// TIA Portal V15.1 export
// export: Created 2024-06-21T08:41:05.5283843Z, ExportSetting WithDefaults, DisplayName Totally Integrated Automation Portal, DisplayVersion V15.1 Update 5, DisplayName TIA Portal Openness, DisplayVersion V15.1 Update 5, DisplayName SINAMICS Startdrive Advanced, DisplayVersion V15.1, DisplayName G130, G150, S120, S150, SINAMICS MV, S210, DisplayVersion V15.1, DisplayName G110M, G120, G120C, G120D, G120P, DisplayVersion V15.1, DisplayName STEP 7 Professional, DisplayVersion V15.1 Update 5, DisplayName STEP 7 Safety, DisplayVersion V15.1, DisplayName WinCC Professional, DisplayVersion V15.1 Update 5, DisplayName SIMATIC Visualization Architect, DisplayVersion V15.1
FUNCTION_BLOCK "LGBMotor2W2S-MoviFitFCPN"   // FB6619, FBD
TITLE = LGBMotor2W2S-MoviFitFCPN
{ S7_Optimized_Access := 'TRUE' }
AUTHOR : ENGIE
FAMILY : Actuator
VERSION : 0.1
// ============================================================================
// This module is used in applications when a Motor 2 way - 2 speed equipped with SEW MOVIFIT FC with fieldbus steering is needed.
// ============================================================================
// stored: AutoNumber false, IsIECCheckEnabled false, IsRetainMemResEnabled false, MemoryReserve 100, SetENOAutomatically False, UDAEnableTagReadback false
   VAR_INPUT
      I_MotorProtection { ExternalAccessible := 'False'; ExternalVisible := 'False'; ExternalWritable := 'False'} : Bool;   // Motor protection
      I_AlarmResetPB { ExternalAccessible := 'False'; ExternalVisible := 'False'; ExternalWritable := 'False'} : Bool;   // Alarm Reset Pushbutton is Activated
      I_SafetyStatusWord { ExternalAccessible := 'False'; ExternalVisible := 'False'; ExternalWritable := 'False'} : Word;   // Safety status word
      I_SafetyControlWord { ExternalAccessible := 'False'; ExternalVisible := 'False'; ExternalWritable := 'False'} : Word;   // Safety control word
      I_SafetyOk { ExternalAccessible := 'False'; ExternalVisible := 'False'; ExternalWritable := 'False'} : Bool;   // Safety ok
      I_MotionStopOk { ExternalAccessible := 'False'; ExternalVisible := 'False'; ExternalWritable := 'False'} : Bool;   // Safety Ok / The motion stop is Ok
      I_LSpdSetMotorCmd { ExternalAccessible := 'False'; ExternalVisible := 'False'; ExternalWritable := 'False'} : Bool;   // Low speed Set Command from function after interlock
      I_HSpdSetMotorCmd { ExternalAccessible := 'False'; ExternalVisible := 'False'; ExternalWritable := 'False'} : Bool;   // High Speed Set Command from function after Interlock
      I_LSpdResMotorCmd { ExternalAccessible := 'False'; ExternalVisible := 'False'; ExternalWritable := 'False'} : Bool;   // Low speed Reset Command from function after interlock
      I_HSpdResMotorCmd { ExternalAccessible := 'False'; ExternalVisible := 'False'; ExternalWritable := 'False'} : Bool;   // High speed Reset Command from function after Interlock
      I_LowSpeed { ExternalAccessible := 'False'; ExternalVisible := 'False'; ExternalWritable := 'False'} : Real;   // Low speed value 0-100%
      I_HighSpeed { ExternalAccessible := 'False'; ExternalVisible := 'False'; ExternalWritable := 'False'} : Real;   // High speed value 0-100%
      I_Ramp { ExternalAccessible := 'False'; ExternalVisible := 'False'; ExternalWritable := 'False'} : Time := T#1s;   // Ramp send in miliseconds (range : 100-10000ms, if 0 then default 1s will be used)
      I_BrakeRelease { ExternalAccessible := 'False'; ExternalVisible := 'False'; ExternalWritable := 'False'} : Bool;   // Command brake release
      I_ParameterSet { ExternalAccessible := 'False'; ExternalVisible := 'False'; ExternalWritable := 'False'} : Bool;   // Select parameter set
   END_VAR
   VAR_OUTPUT
      O_MotorProtectionAlarm { ExternalAccessible := 'False'; ExternalVisible := 'False'; ExternalWritable := 'False'} : Bool;   // Motor protection alarm
      O_SafetySwitchAlarm { ExternalAccessible := 'False'; ExternalVisible := 'False'; ExternalWritable := 'False'} : Bool;   // Safety switch alarm
      O_ConfigRampAlarm { ExternalAccessible := 'False'; ExternalVisible := 'False'; ExternalWritable := 'False'} : Bool;   // Config alarm
      O_ConfigRampCalcAlarm { ExternalAccessible := 'False'; ExternalVisible := 'False'; ExternalWritable := 'False'} : Bool;   // Config alarm
      O_STOAlarm { ExternalAccessible := 'False'; ExternalVisible := 'False'; ExternalWritable := 'False'} : Bool;   // Drive fault / STO alarm
      O_MotionStopWarning { ExternalAccessible := 'False'; ExternalVisible := 'False'; ExternalWritable := 'False'} : Bool;   // Drive fault / Motion Stop warning
      O_DriveFaultAlarm { ExternalAccessible := 'False'; ExternalVisible := 'False'; ExternalWritable := 'False'} : Bool;   // Drive fault
      O_DriveWarning { ExternalAccessible := 'False'; ExternalVisible := 'False'; ExternalWritable := 'False'} : Bool;   // Drive warning
      O_DriveReady { ExternalAccessible := 'False'; ExternalVisible := 'False'; ExternalWritable := 'False'} : Bool;   // Drive ready
      O_PODataNotEnabled { ExternalAccessible := 'False'; ExternalVisible := 'False'; ExternalWritable := 'False'} : Bool;   // Process data is enabled (1 = Drive can be controlled via fieldbus)
      O_ParameterSet { ExternalAccessible := 'False'; ExternalVisible := 'False'; ExternalWritable := 'False'} : Bool;   // Active parameter set
      O_OutputStageEnabled { ExternalAccessible := 'False'; ExternalVisible := 'False'; ExternalWritable := 'False'} : Bool;   // Inverter output stage is enabled
      O_Brake { ExternalAccessible := 'False'; ExternalVisible := 'False'; ExternalWritable := 'False'} : Bool;   // Brake status
      O_AlarmABCondition { ExternalAccessible := 'False'; ExternalVisible := 'False'; ExternalWritable := 'False'} : Bool;   // Alarm AB Condition
   END_VAR
   VAR_IN_OUT
      IO_Modes : "Modes";
      IO_Alarm : "Alarm";
      H_HMI : "H_HMI";
      "H_GBMotor2W2S-MoviFitFCPN" : "H_GBMotor2W2S-MoviFitFCPN";   // HMI UDT
      C_EnableAlarm { ExternalAccessible := 'False'; ExternalVisible := 'False'; ExternalWritable := 'False'} : Bool;   // Enable Alarm
      C_MotorProtectionUsed { ExternalAccessible := 'False'; ExternalVisible := 'False'; ExternalWritable := 'False'} : Bool := True;   // Motor Protection used
      C_MotorProtectionNc { ExternalAccessible := 'False'; ExternalVisible := 'False'; ExternalWritable := 'False'} : Bool := True;   // Motor Protection Normally closed
      C_MotionStopUsed { ExternalAccessible := 'False'; ExternalVisible := 'False'; ExternalWritable := 'False'} : Bool;   // Motion Stop used
      C_HWSubInput { ExternalAccessible := 'False'; ExternalVisible := 'False'; ExternalWritable := 'False'} : HW_SUBMODULE;   // Inputs telegram 3 Hardware identifier
      C_HWSubInputStatus { ExternalAccessible := 'False'; ExternalVisible := 'False'; ExternalWritable := 'False'} : HW_SUBMODULE;   // Status telegram MOVIFIT Hardware identifier
      C_HWSubOutput { ExternalAccessible := 'False'; ExternalVisible := 'False'; ExternalWritable := 'False'} : HW_SUBMODULE;   // Outputs telegram 3 Hardware identifier
      C_InitDirection { ExternalAccessible := 'False'; ExternalVisible := 'False'; ExternalWritable := 'False'} : Bool;   // Initialisation of the direction
      C_DriveCurrent { ExternalAccessible := 'False'; ExternalVisible := 'False'; ExternalWritable := 'False'} : Real;   // Reference current of the drive
      C_MotorCurrent { ExternalAccessible := 'False'; ExternalVisible := 'False'; ExternalWritable := 'False'} : Real;   // Reference current of the motor
      C_MotorRPM { ExternalAccessible := 'False'; ExternalVisible := 'False'; ExternalWritable := 'False'} : Real;   // Reference RPM of the motor
      C_RatioGearbox { ExternalAccessible := 'False'; ExternalVisible := 'False'; ExternalWritable := 'False'} : Real;   // Ratio Gearbox <-> Motor
      C_Diameter { ExternalAccessible := 'False'; ExternalVisible := 'False'; ExternalWritable := 'False'} : Real;   // Diameter in mm
      C_Acceleration { ExternalAccessible := 'False'; ExternalVisible := 'False'; ExternalWritable := 'False'} : Real;   // Acceleration in m/s²
   END_VAR
   VAR
      EnableAlarmHWSR { ExternalAccessible := 'False'; ExternalVisible := 'False'; ExternalWritable := 'False'} : Bool;   // Enable Alarms from the hardware
      EnableAlarmHW { ExternalAccessible := 'False'; ExternalVisible := 'False'; ExternalWritable := 'False'} : Bool;   // Enable Alarms from the hardware
      SetFrequency { ExternalAccessible := 'False'; ExternalVisible := 'False'; ExternalWritable := 'False'} : Real;   // Set frequency dependant on config
      ResFrequency { ExternalAccessible := 'False'; ExternalVisible := 'False'; ExternalWritable := 'False'} : Real;   // Reset frequency dependant on config
      MotorProtectionAlarm { ExternalAccessible := 'False'; ExternalVisible := 'False'; ExternalWritable := 'False'} : Bool;   // Motor protection alarm
      MotorProtectionAlarmABCond { ExternalAccessible := 'False'; ExternalVisible := 'False'; ExternalWritable := 'False'} : Bool;   // Motor protection alarm condition
      SafetySwitchAlarm { ExternalAccessible := 'False'; ExternalVisible := 'False'; ExternalWritable := 'False'} : Bool;   // Safety Switch alarm
      SafetySwitchAlarmABCond { ExternalAccessible := 'False'; ExternalVisible := 'False'; ExternalWritable := 'False'} : Bool;   // Safety Switch alarm condition
      DriveFaultAlarm { ExternalAccessible := 'False'; ExternalVisible := 'False'; ExternalWritable := 'False'} : Bool;   // Drive fault alarm
      DriveFaultAlarmABCond { ExternalAccessible := 'False'; ExternalVisible := 'False'; ExternalWritable := 'False'} : Bool;   // Drive fault alarm condition
      STOAlarm { ExternalAccessible := 'False'; ExternalVisible := 'False'; ExternalWritable := 'False'} : Bool;   // Drive fault alarm / STO feedback fault alarm
      STOAlarmABCond { ExternalAccessible := 'False'; ExternalVisible := 'False'; ExternalWritable := 'False'} : Bool;   // Drive fault alarm condition / STO feedback fault alarm condition
      MotionStopWarning { ExternalAccessible := 'False'; ExternalVisible := 'False'; ExternalWritable := 'False'} : Bool;   // Drive fault alarm / Motion Stop warning
      ConfigRampAlarm { ExternalAccessible := 'False'; ExternalVisible := 'False'; ExternalWritable := 'False'} : Bool;   // Config alarm
      ConfigRampCalcAlarm { ExternalAccessible := 'False'; ExternalVisible := 'False'; ExternalWritable := 'False'} : Bool;   // Config alarm
      Start { ExternalAccessible := 'False'; ExternalVisible := 'False'; ExternalWritable := 'False'} : Bool;   // Start command to drive
      SetpointSpeed { ExternalAccessible := 'False'; ExternalVisible := 'False'; ExternalWritable := 'False'} : Real;   // Setpoint speed
      SetpointSpeedCalc { ExternalAccessible := 'False'; ExternalVisible := 'False'; ExternalWritable := 'False'} : Real;   // Setpoint speed
      OutputStageEnabled { ExternalAccessible := 'False'; ExternalVisible := 'False'; ExternalWritable := 'False'} : Bool;   // Inverter output stage is enabled
      MaintenanceSwitch { ExternalAccessible := 'False'; ExternalVisible := 'False'; ExternalWritable := 'False'} : Bool;   // Maintenance switch activated (1=mains OFF)
      PODataEnabled { ExternalAccessible := 'False'; ExternalVisible := 'False'; ExternalWritable := 'False'} : Bool;   // Process data is enabled (1 = Drive can be controlled via fieldbus)
      PODataDisabled { ExternalAccessible := 'False'; ExternalVisible := 'False'; ExternalWritable := 'False'} : Bool;   // Process data is enabled (1 = Drive can be controlled via fieldbus)
      Fault { ExternalAccessible := 'False'; ExternalVisible := 'False'; ExternalWritable := 'False'} : Bool;   // Fault present
      Brake { ExternalAccessible := 'False'; ExternalVisible := 'False'; ExternalWritable := 'False'} : Bool;   // Brake status
      ActorVoltageOverloadDO00 { ExternalAccessible := 'False'; ExternalVisible := 'False'; ExternalWritable := 'False'} : Bool;   // Short circuit / overload of the actuator voltage for digital output DO00
      ActorVoltageOverloadDO01 { ExternalAccessible := 'False'; ExternalVisible := 'False'; ExternalWritable := 'False'} : Bool;   // Short circuit / overload of the actuator voltage for digital output DO01
      ActorVoltageOverloadDO02 { ExternalAccessible := 'False'; ExternalVisible := 'False'; ExternalWritable := 'False'} : Bool;   // Short circuit / overload of the actuator voltage for digital output DO02
      ActorVoltageOverloadDO03 { ExternalAccessible := 'False'; ExternalVisible := 'False'; ExternalWritable := 'False'} : Bool;   // Short circuit / overload of the actuator voltage for digital output DO03
      SensorVoltageOverloadGroup1 { ExternalAccessible := 'False'; ExternalVisible := 'False'; ExternalWritable := 'False'} : Bool;   // Short circuit / overload of the sensor suuply group 1 (VO24-I)
      SensorVoltageOverloadGroup2 { ExternalAccessible := 'False'; ExternalVisible := 'False'; ExternalWritable := 'False'} : Bool;   // Short circuit / overload of the sensor suuply group 2 (VO24-I)
      SensorVoltageOverloadGroup3 { ExternalAccessible := 'False'; ExternalVisible := 'False'; ExternalWritable := 'False'} : Bool;   // Short circuit / overload of the sensor suuply group 3 (VO24-I)
      SensorVoltageOverloadGroup4 { ExternalAccessible := 'False'; ExternalVisible := 'False'; ExternalWritable := 'False'} : Bool;   // Short circuit / overload of the sensor suuply group 4 (VO24-I)
      "Undervoltage24V-S" { ExternalAccessible := 'False'; ExternalVisible := 'False'; ExternalWritable := 'False'} : Bool;   // Value falls below the power limit for the actuator voltage DO00-03
      "InverterVoltageNotApplied24V-P" { ExternalAccessible := 'False'; ExternalVisible := 'False'; ExternalWritable := 'False'} : Bool;   // Presence of 24V_P for integrated inverter (FC) or external MOVIMOT (1=24V_P not present)
      MOVIFITSystemFault { ExternalAccessible := 'False'; ExternalVisible := 'False'; ExternalWritable := 'False'} : Bool;   // MOVIFIT system fault
      RampToDrive { ExternalAccessible := 'False'; ExternalVisible := 'False'; ExternalWritable := 'False'} : Time;   // Calculated Ramp send in miliseconds
      _MoviFitPN { ExternalAccessible := 'False'; ExternalVisible := 'False'; ExternalWritable := 'False'} : "LGBSEW-MoviFitFCPN";   // SEW MOVIFIT FC
      _MotorProtection { ExternalAccessible := 'False'; ExternalVisible := 'False'; ExternalWritable := 'False'} : "L1AlarmMultiIn";   // FB
      _SafetySwitch { ExternalAccessible := 'False'; ExternalVisible := 'False'; ExternalWritable := 'False'} : "L1AlarmMultiIn";   // FB
      _DriveFault { ExternalAccessible := 'False'; ExternalVisible := 'False'; ExternalWritable := 'False'} : "L1AlarmMultiIn";   // FB
      _STO { ExternalAccessible := 'False'; ExternalVisible := 'False'; ExternalWritable := 'False'} : "L1AlarmMultiIn";   // FB
      _MotionStop { ExternalAccessible := 'False'; ExternalVisible := 'False'; ExternalWritable := 'False'} : "L1AlarmMultiIn";   // FB
      T_STOAlarm { ExternalAccessible := 'False'; ExternalVisible := 'False'; ExternalWritable := 'False'} : TON_TIME;   // Timer
      T_Reboot { ExternalAccessible := 'False'; ExternalVisible := 'False'; ExternalWritable := 'False'} : TON_TIME;   // Timer / Timer Reboot
   END_VAR
   VAR_TEMP   // added for the SCL form of the ladder/FBD networks
      _w1 : Bool;
   END_VAR
BEGIN

REGION Network 1: **** 2.1 - Alarms - Enable Alarms **** Enable Hardware Alarm
   // Enable Hardware Alarm
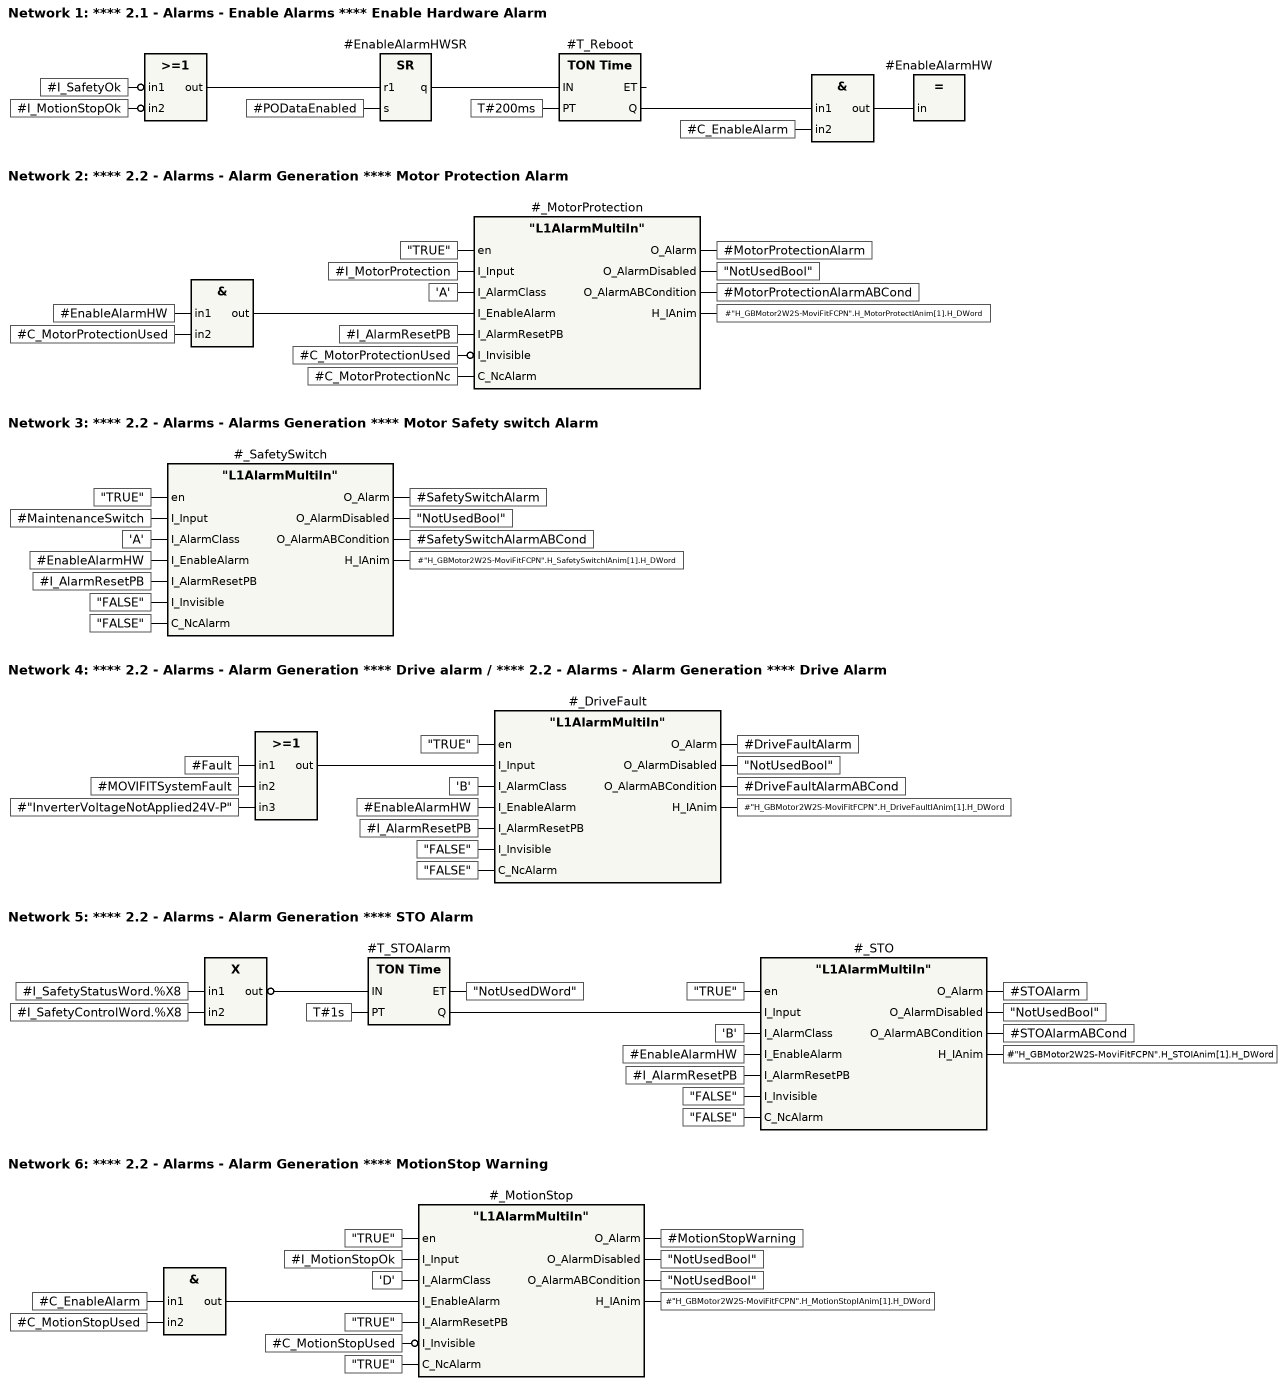
   IF #PODataEnabled THEN
       #EnableAlarmHWSR := TRUE;   // SR flip-flop
   END_IF;
   IF NOT #I_SafetyOk OR NOT #I_MotionStopOk THEN #EnableAlarmHWSR := FALSE; END_IF;
   #T_Reboot(IN := #EnableAlarmHWSR, PT := T#200ms);   // TON
   #EnableAlarmHW := #T_Reboot.Q AND #C_EnableAlarm;
END_REGION

REGION Network 2: **** 2.2 - Alarms - Alarm Generation **** Motor Protection Alarm
   // Motor Protection Alarm
   IF "TRUE" THEN
       #_MotorProtection(I_Input := #I_MotorProtection,   // "L1AlarmMultiIn"
                         I_AlarmClass := 'A',
                         I_EnableAlarm := #EnableAlarmHW AND #C_MotorProtectionUsed,
                         I_AlarmResetPB := #I_AlarmResetPB,
                         I_Invisible := NOT #C_MotorProtectionUsed,
                         C_NcAlarm := #C_MotorProtectionNc,
                         O_Alarm => #MotorProtectionAlarm,
                         O_AlarmDisabled => "NotUsedBool",
                         O_AlarmABCondition => #MotorProtectionAlarmABCond,
                         H_IAnim => #"H_GBMotor2W2S-MoviFitFCPN".H_MotorProtectIAnim[1].H_DWord);
   END_IF;
END_REGION

REGION Network 3: **** 2.2 - Alarms - Alarms Generation **** Motor Safety switch Alarm
   // Motor Safety switch Alarm
   IF "TRUE" THEN
       #_SafetySwitch(I_Input := #MaintenanceSwitch,   // "L1AlarmMultiIn"
                      I_AlarmClass := 'A',
                      I_EnableAlarm := #EnableAlarmHW,
                      I_AlarmResetPB := #I_AlarmResetPB,
                      I_Invisible := "FALSE",
                      C_NcAlarm := "FALSE",
                      O_Alarm => #SafetySwitchAlarm,
                      O_AlarmDisabled => "NotUsedBool",
                      O_AlarmABCondition => #SafetySwitchAlarmABCond,
                      H_IAnim => #"H_GBMotor2W2S-MoviFitFCPN".H_SafetySwitchIAnim[1].H_DWord);
   END_IF;
END_REGION

REGION Network 4: **** 2.2 - Alarms - Alarm Generation **** Drive alarm / **** 2.2 - Alarms - Alarm Generation **** Drive Alarm
   IF "TRUE" THEN
       #_DriveFault(I_Input := #Fault OR #MOVIFITSystemFault OR #"InverterVoltageNotApplied24V-P",   // "L1AlarmMultiIn"
                    I_AlarmClass := 'B',
                    I_EnableAlarm := #EnableAlarmHW,
                    I_AlarmResetPB := #I_AlarmResetPB,
                    I_Invisible := "FALSE",
                    C_NcAlarm := "FALSE",
                    O_Alarm => #DriveFaultAlarm,
                    O_AlarmDisabled => "NotUsedBool",
                    O_AlarmABCondition => #DriveFaultAlarmABCond,
                    H_IAnim => #"H_GBMotor2W2S-MoviFitFCPN".H_DriveFaultIAnim[1].H_DWord);
   END_IF;
END_REGION

REGION Network 5: **** 2.2 - Alarms - Alarm Generation **** STO Alarm
   #T_STOAlarm(IN := NOT (#I_SafetyStatusWord.%X8 XOR #I_SafetyControlWord.%X8),   // TON
               PT := T#1s,
               ET => "NotUsedDWord");
   IF "TRUE" THEN
       #_STO(I_Input := #T_STOAlarm.Q,   // "L1AlarmMultiIn"
             I_AlarmClass := 'B',
             I_EnableAlarm := #EnableAlarmHW,
             I_AlarmResetPB := #I_AlarmResetPB,
             I_Invisible := "FALSE",
             C_NcAlarm := "FALSE",
             O_Alarm => #STOAlarm,
             O_AlarmDisabled => "NotUsedBool",
             O_AlarmABCondition => #STOAlarmABCond,
             H_IAnim => #"H_GBMotor2W2S-MoviFitFCPN".H_STOIAnim[1].H_DWord);
   END_IF;
END_REGION

REGION Network 6: **** 2.2 - Alarms - Alarm Generation **** MotionStop Warning
   IF "TRUE" THEN
       #_MotionStop(I_Input := #I_MotionStopOk,   // "L1AlarmMultiIn"
                    I_AlarmClass := 'D',
                    I_EnableAlarm := #C_EnableAlarm AND #C_MotionStopUsed,
                    I_AlarmResetPB := "TRUE",
                    I_Invisible := NOT #C_MotionStopUsed,
                    C_NcAlarm := "TRUE",
                    O_Alarm => #MotionStopWarning,
                    O_AlarmDisabled => "NotUsedBool",
                    O_AlarmABCondition => "NotUsedBool",
                    H_IAnim => #"H_GBMotor2W2S-MoviFitFCPN".H_MotionStopIAnim[1].H_DWord);
   END_IF;
END_REGION

REGION Network 7: **** 2.2 - Alarms - Alarm Generation **** PO data not enabled
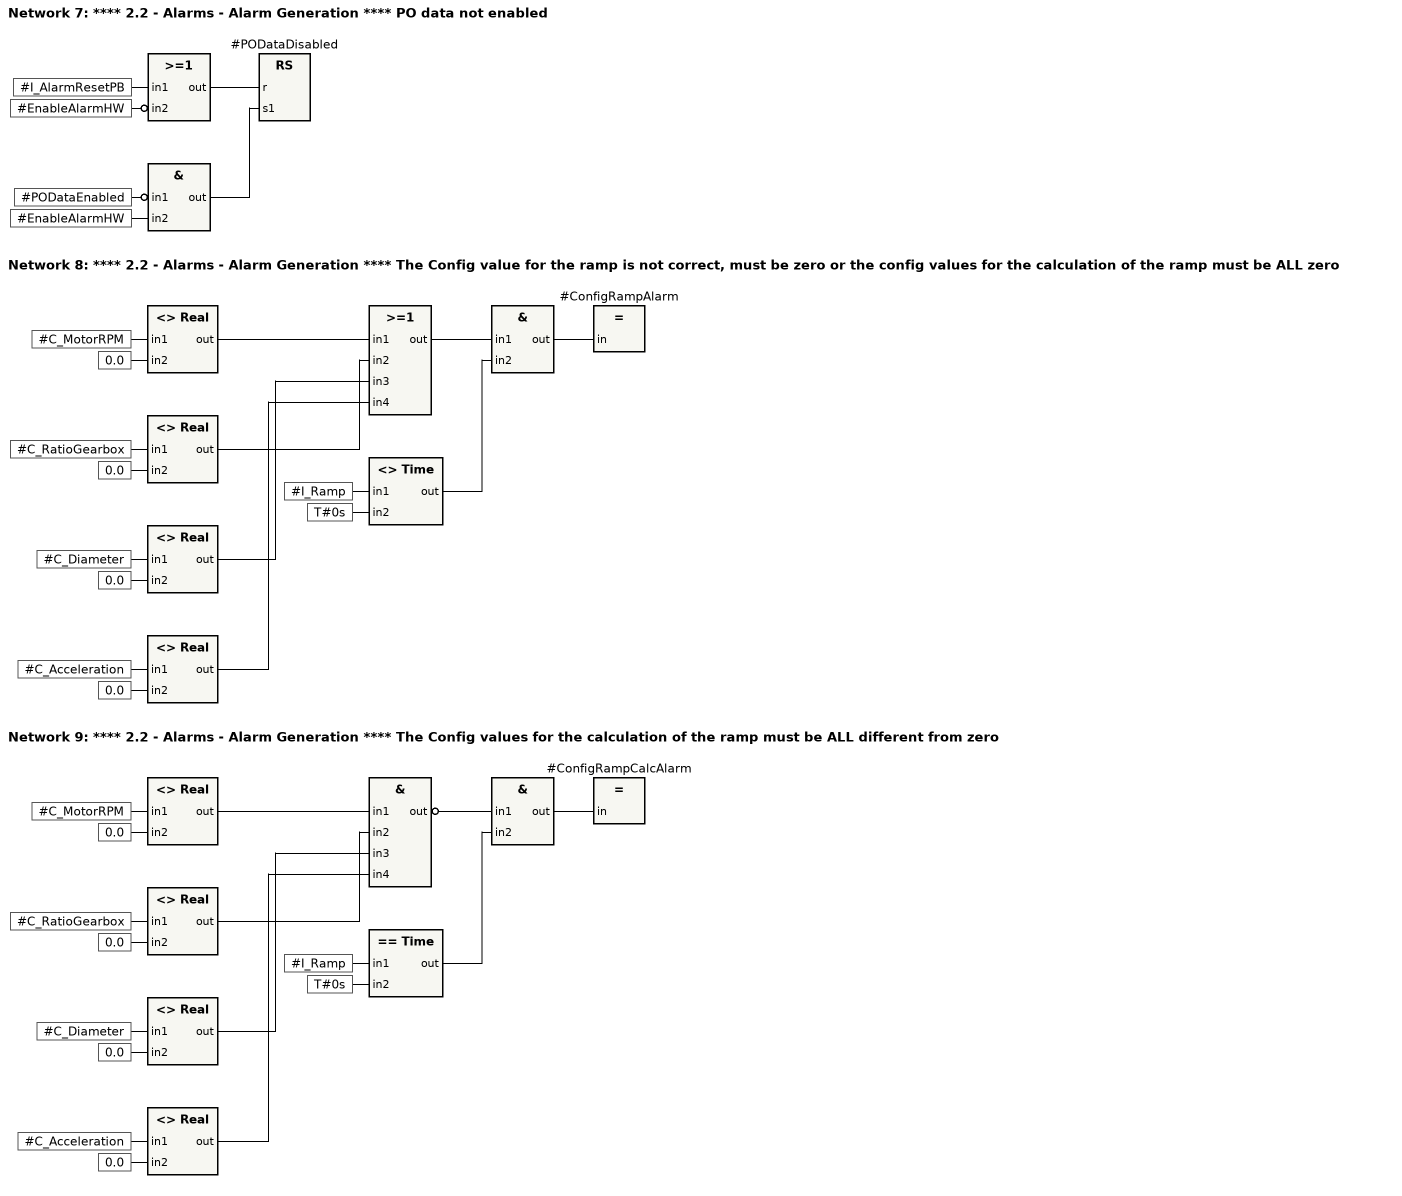
   IF #I_AlarmResetPB OR NOT #EnableAlarmHW THEN
       #PODataDisabled := FALSE;   // RS flip-flop
   END_IF;
   IF NOT #PODataEnabled AND #EnableAlarmHW THEN #PODataDisabled := TRUE; END_IF;
END_REGION

REGION Network 8: **** 2.2 - Alarms - Alarm Generation **** The Config value for the ramp is not correct, must be zero or the config values for the calculation of the ramp must be ALL zero
   #ConfigRampAlarm := ((#C_MotorRPM <> 0.0) OR (#C_RatioGearbox <> 0.0) OR (#C_Diameter <> 0.0) OR (#C_Acceleration <> 0.0)) AND (#I_Ramp <> T#0s);
END_REGION

REGION Network 9: **** 2.2 - Alarms - Alarm Generation **** The Config values for the calculation of the ramp must be ALL different from zero
   #ConfigRampCalcAlarm := NOT ((#C_MotorRPM <> 0.0) AND (#C_RatioGearbox <> 0.0) AND (#C_Diameter <> 0.0) AND (#C_Acceleration <> 0.0)) AND (#I_Ramp = T#0s);
END_REGION

REGION Network 10: **** 4.6 - Machine Status - Indication **** Icon Animation
   // Icon Animation
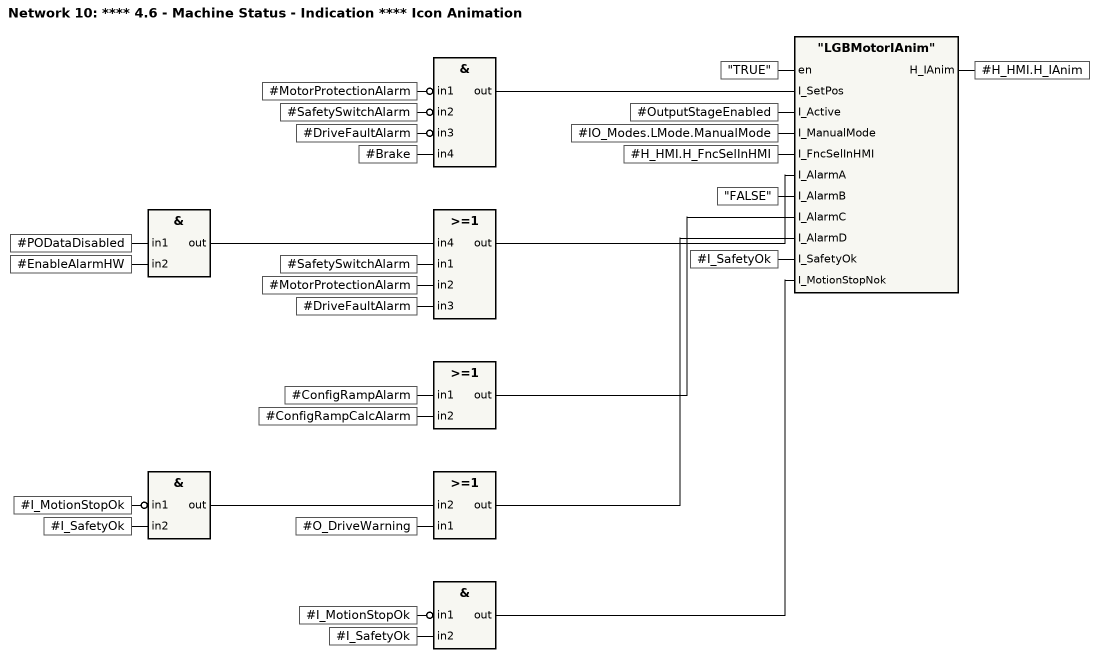
   IF "TRUE" THEN
       "LGBMotorIAnim"(I_SetPos := NOT #MotorProtectionAlarm AND NOT #SafetySwitchAlarm AND NOT #DriveFaultAlarm AND #Brake,
                       I_Active := #OutputStageEnabled,
                       I_ManualMode := #IO_Modes.LMode.ManualMode,
                       I_FncSelInHMI := #H_HMI.H_FncSelInHMI,
                       I_AlarmA := (#PODataDisabled AND #EnableAlarmHW) OR #SafetySwitchAlarm OR #MotorProtectionAlarm OR #DriveFaultAlarm,
                       I_AlarmB := "FALSE",
                       I_AlarmC := #ConfigRampAlarm OR #ConfigRampCalcAlarm,
                       I_AlarmD := (NOT #I_MotionStopOk AND #I_SafetyOk) OR #O_DriveWarning,
                       I_SafetyOk := #I_SafetyOk,
                       I_MotionStopNok := NOT #I_MotionStopOk AND #I_SafetyOk,
                       H_IAnim => #H_HMI.H_IAnim);
   END_IF;
END_REGION

REGION Network 11: **** 4.6 - Machine Status - Indication **** Animation
   // Animation
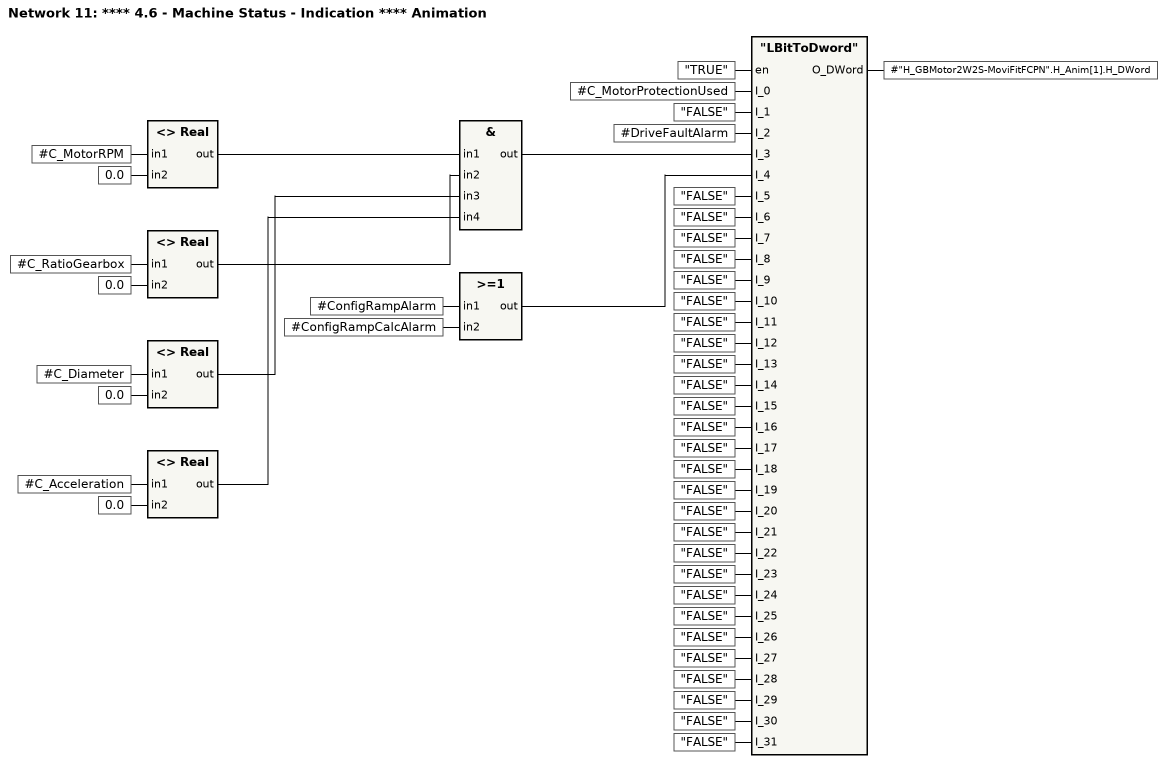
   IF "TRUE" THEN
       "LBitToDword"(I_0 := #C_MotorProtectionUsed,
                     I_1 := "FALSE",
                     I_2 := #DriveFaultAlarm,
                     I_3 := (#C_MotorRPM <> 0.0) AND (#C_RatioGearbox <> 0.0) AND (#C_Diameter <> 0.0) AND (#C_Acceleration <> 0.0),
                     I_4 := #ConfigRampAlarm OR #ConfigRampCalcAlarm,
                     I_5 := "FALSE",
                     I_6 := "FALSE",
                     I_7 := "FALSE",
                     I_8 := "FALSE",
                     I_9 := "FALSE",
                     I_10 := "FALSE",
                     I_11 := "FALSE",
                     I_12 := "FALSE",
                     I_13 := "FALSE",
                     I_14 := "FALSE",
                     I_15 := "FALSE",
                     I_16 := "FALSE",
                     I_17 := "FALSE",
                     I_18 := "FALSE",
                     I_19 := "FALSE",
                     I_20 := "FALSE",
                     I_21 := "FALSE",
                     I_22 := "FALSE",
                     I_23 := "FALSE",
                     I_24 := "FALSE",
                     I_25 := "FALSE",
                     I_26 := "FALSE",
                     I_27 := "FALSE",
                     I_28 := "FALSE",
                     I_29 := "FALSE",
                     I_30 := "FALSE",
                     I_31 := "FALSE",
                     O_DWord => #"H_GBMotor2W2S-MoviFitFCPN".H_Anim[1].H_DWord);
   END_IF;
END_REGION

REGION Network 12: **** 4.6 - Machine Status - Indication **** Safety words
   // Animation
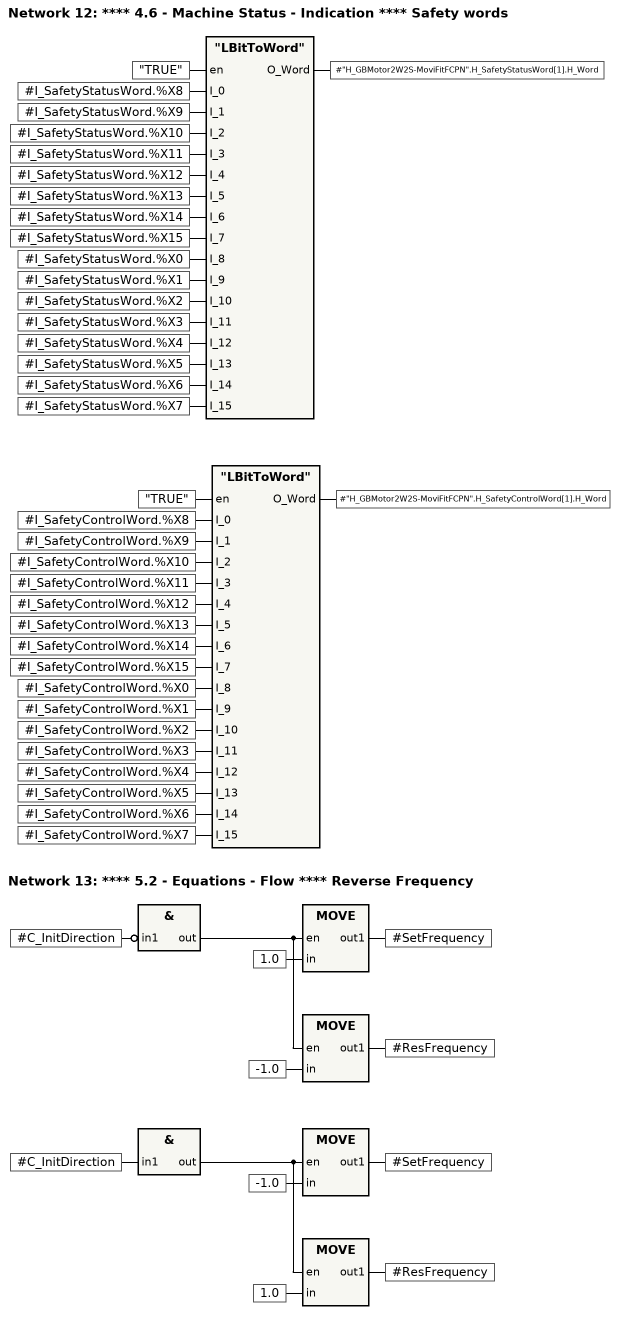
   IF "TRUE" THEN
       "LBitToWord"(I_0 := #I_SafetyStatusWord.%X8,
                    I_1 := #I_SafetyStatusWord.%X9,
                    I_2 := #I_SafetyStatusWord.%X10,
                    I_3 := #I_SafetyStatusWord.%X11,
                    I_4 := #I_SafetyStatusWord.%X12,
                    I_5 := #I_SafetyStatusWord.%X13,
                    I_6 := #I_SafetyStatusWord.%X14,
                    I_7 := #I_SafetyStatusWord.%X15,
                    I_8 := #I_SafetyStatusWord.%X0,
                    I_9 := #I_SafetyStatusWord.%X1,
                    I_10 := #I_SafetyStatusWord.%X2,
                    I_11 := #I_SafetyStatusWord.%X3,
                    I_12 := #I_SafetyStatusWord.%X4,
                    I_13 := #I_SafetyStatusWord.%X5,
                    I_14 := #I_SafetyStatusWord.%X6,
                    I_15 := #I_SafetyStatusWord.%X7,
                    O_Word => #"H_GBMotor2W2S-MoviFitFCPN".H_SafetyStatusWord[1].H_Word);
   END_IF;
   IF "TRUE" THEN
       "LBitToWord"(I_0 := #I_SafetyControlWord.%X8,
                    I_1 := #I_SafetyControlWord.%X9,
                    I_2 := #I_SafetyControlWord.%X10,
                    I_3 := #I_SafetyControlWord.%X11,
                    I_4 := #I_SafetyControlWord.%X12,
                    I_5 := #I_SafetyControlWord.%X13,
                    I_6 := #I_SafetyControlWord.%X14,
                    I_7 := #I_SafetyControlWord.%X15,
                    I_8 := #I_SafetyControlWord.%X0,
                    I_9 := #I_SafetyControlWord.%X1,
                    I_10 := #I_SafetyControlWord.%X2,
                    I_11 := #I_SafetyControlWord.%X3,
                    I_12 := #I_SafetyControlWord.%X4,
                    I_13 := #I_SafetyControlWord.%X5,
                    I_14 := #I_SafetyControlWord.%X6,
                    I_15 := #I_SafetyControlWord.%X7,
                    O_Word => #"H_GBMotor2W2S-MoviFitFCPN".H_SafetyControlWord[1].H_Word);
   END_IF;
END_REGION

REGION Network 13: **** 5.2 - Equations - Flow **** Reverse Frequency
   // Reverse frequency dependant on config
   IF NOT #C_InitDirection THEN
       #SetFrequency := 1.0;
       #ResFrequency := -1.0;
   END_IF;
   IF #C_InitDirection THEN
       #SetFrequency := -1.0;
       #ResFrequency := 1.0;
   END_IF;
END_REGION

REGION Network 14: **** 5.2 - Equations - Flow Equations **** High speed setting to drive / **** 5.2 - Equations - Flow Equations **** High speed Setpoint Speed to drive
   // Select high speed
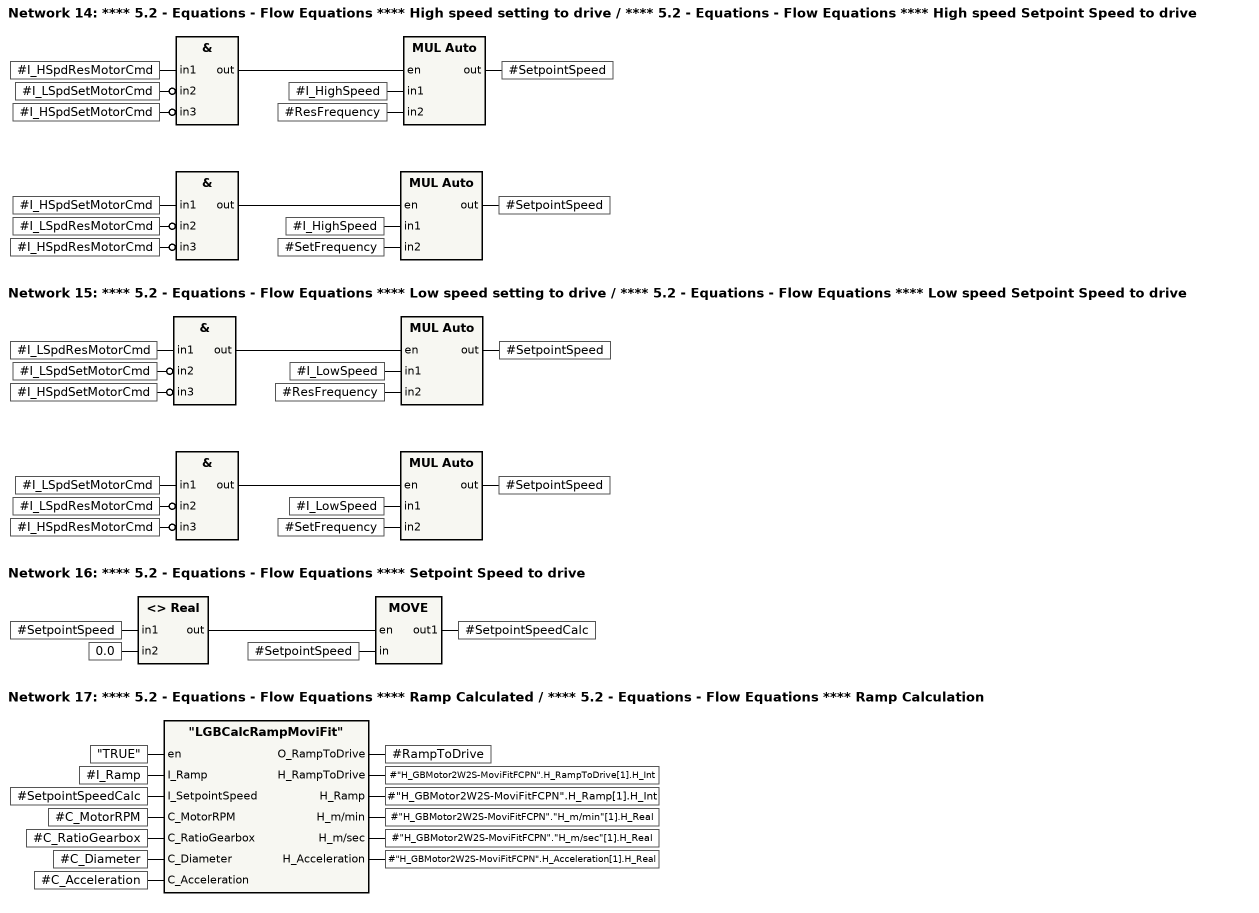
   IF #I_HSpdResMotorCmd AND NOT #I_LSpdSetMotorCmd AND NOT #I_HSpdSetMotorCmd THEN
       #SetpointSpeed := #I_HighSpeed * #ResFrequency;
   END_IF;
   IF #I_HSpdSetMotorCmd AND NOT #I_LSpdResMotorCmd AND NOT #I_HSpdResMotorCmd THEN
       #SetpointSpeed := #I_HighSpeed * #SetFrequency;
   END_IF;
END_REGION

REGION Network 15: **** 5.2 - Equations - Flow Equations **** Low speed setting to drive / **** 5.2 - Equations - Flow Equations **** Low speed Setpoint Speed to drive
   IF #I_LSpdResMotorCmd AND NOT #I_LSpdSetMotorCmd AND NOT #I_HSpdSetMotorCmd THEN
       #SetpointSpeed := #I_LowSpeed * #ResFrequency;
   END_IF;
   IF #I_LSpdSetMotorCmd AND NOT #I_LSpdResMotorCmd AND NOT #I_HSpdResMotorCmd THEN
       #SetpointSpeed := #I_LowSpeed * #SetFrequency;
   END_IF;
END_REGION

REGION Network 16: **** 5.2 - Equations - Flow Equations **** Setpoint Speed to drive
   IF #SetpointSpeed <> 0.0 THEN #SetpointSpeedCalc := #SetpointSpeed; END_IF;
END_REGION

REGION Network 17: **** 5.2 - Equations - Flow Equations **** Ramp Calculated / **** 5.2 - Equations - Flow Equations **** Ramp Calculation
   IF "TRUE" THEN
       "LGBCalcRampMoviFit"(I_Ramp := #I_Ramp,
                            I_SetpointSpeed := #SetpointSpeedCalc,
                            C_MotorRPM := #C_MotorRPM,
                            C_RatioGearbox := #C_RatioGearbox,
                            C_Diameter := #C_Diameter,
                            C_Acceleration := #C_Acceleration,
                            O_RampToDrive => #RampToDrive,
                            H_RampToDrive => #"H_GBMotor2W2S-MoviFitFCPN".H_RampToDrive[1].H_Int,
                            H_Ramp => #"H_GBMotor2W2S-MoviFitFCPN".H_Ramp[1].H_Int,
                            "H_m/min" => #"H_GBMotor2W2S-MoviFitFCPN"."H_m/min"[1].H_Real,
                            "H_m/sec" => #"H_GBMotor2W2S-MoviFitFCPN"."H_m/sec"[1].H_Real,
                            H_Acceleration => #"H_GBMotor2W2S-MoviFitFCPN".H_Acceleration[1].H_Real);
   END_IF;
END_REGION

REGION Network 18: **** 5.2 - Equations - Flow Equations **** Start command to drive
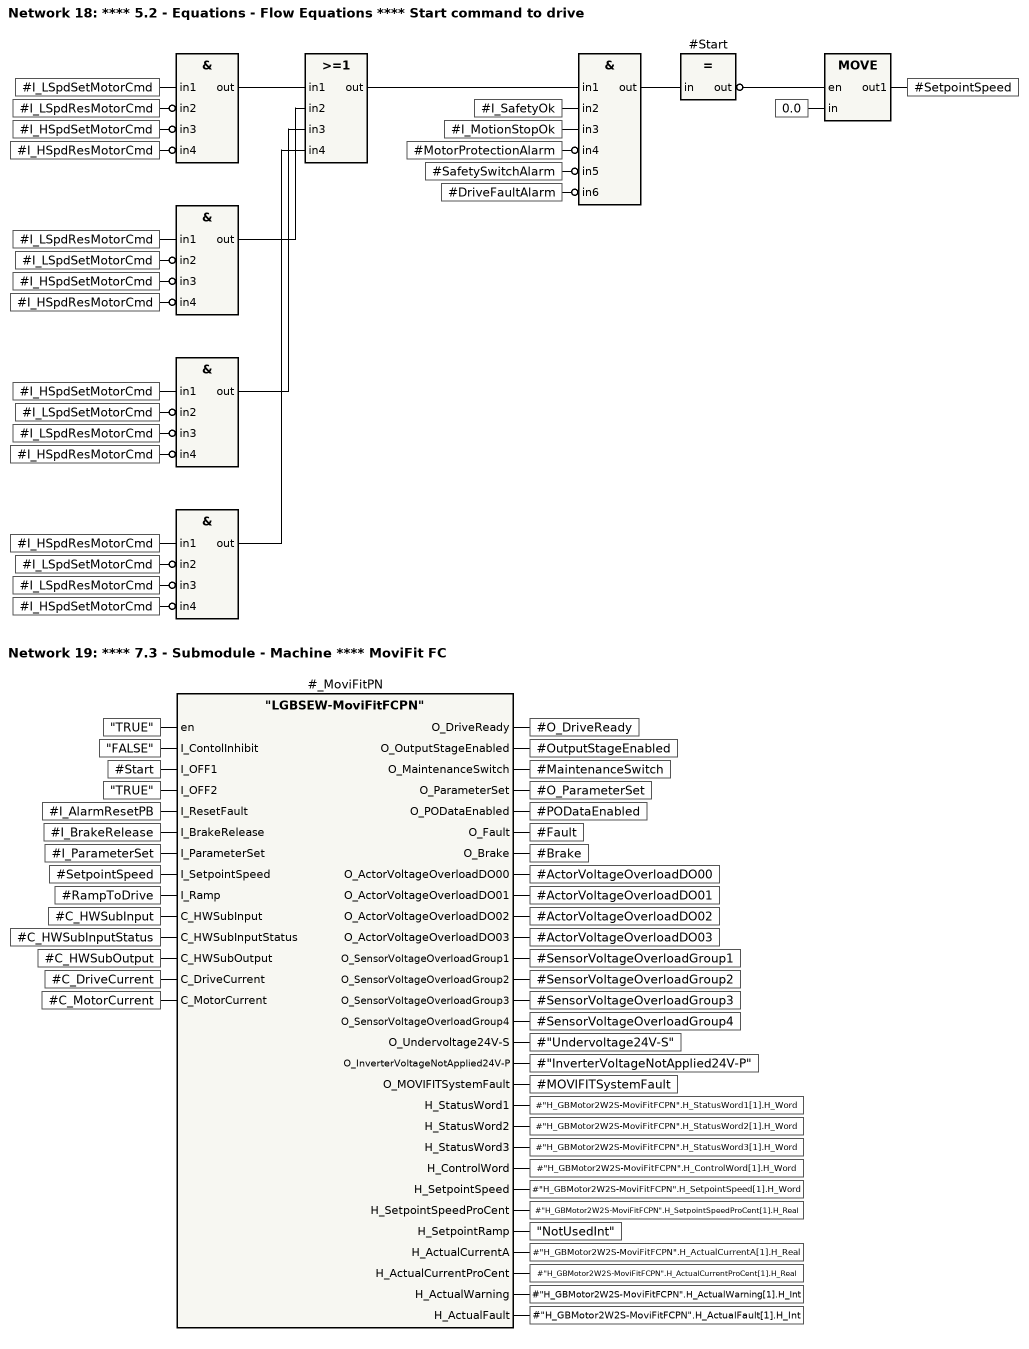
   #_w1 := ((#I_LSpdSetMotorCmd AND NOT #I_LSpdResMotorCmd AND NOT #I_HSpdSetMotorCmd AND NOT #I_HSpdResMotorCmd) OR (#I_LSpdResMotorCmd AND NOT #I_LSpdSetMotorCmd AND NOT #I_HSpdSetMotorCmd AND NOT #I_HSpdResMotorCmd) OR (#I_HSpdSetMotorCmd AND NOT #I_LSpdSetMotorCmd AND NOT #I_LSpdResMotorCmd AND NOT #I_HSpdResMotorCmd) OR (#I_HSpdResMotorCmd AND NOT #I_LSpdSetMotorCmd AND NOT #I_LSpdResMotorCmd AND NOT #I_HSpdSetMotorCmd)) AND #I_SafetyOk AND #I_MotionStopOk AND NOT #MotorProtectionAlarm AND NOT #SafetySwitchAlarm AND NOT #DriveFaultAlarm;
   #Start := #_w1;   // Only 1 of the 4 commands may be active or else there is no start commend, if there is no start command the setpoint for the drive is also 0%
   IF NOT #_w1 THEN #SetpointSpeed := 0.0; END_IF;
END_REGION

REGION Network 19: **** 7.3 - Submodule - Machine **** MoviFit FC
   IF "TRUE" THEN
       #_MoviFitPN(I_ContolInhibit := "FALSE",   // "LGBSEW-MoviFitFCPN": Copy data with HW ID _________ /________ / l input telegram l SEW l l ===============>> PLC l Drive _l / <<=============== -l__l output telegram ********************************************************** SEW drive config: - 8.. Unit functions l - 87 Process data assignment _____________________ 870 Setpoint description PO1 l Control word 2 v l _____________________ 871 Setpoint description PO2 l Setpoint speed [%] v l _____________________ 872 Setpoint description PO3 l Ramp v l _____________________ 873 Actual value description PI1 l Status word 1 v l _____________________ 874 Actual value description PI2 l Output current v l _____________________ 875 Actual value description PI3 l Status word 2 v l _____________________ 876 PO data enable l Yes v l l v This changes to no when a POx paramater is changed Dot not forget to put this back to yes ! ********************************************************** "I_Ramp" is send to the drive in ms. Speed The ramp up / down time is (Rpm) ^ / set with this parameter l _________ / l / \/ l / \ l____/ \____ l--------------------------------------------------> t (s) _ ********************************************************** "I_OFF1" & "I_OFF2" example: ^ Speed (%) Stop signal at 5s l / 100% l______________/_ l \ \ l \ \ l \ \ l \ \ 0% l___________________\_____\___________________________> Time (s) l OFF2 OFF1 (regular start stop) 7s 10s Ramp down time settings to be done in the drive. OFF2 is to be used for controlled stops when there is a need to stop faster then regular, for example when there is an E-stop at a lift it is better to do a controlled stop and after that (x time in safety program) to give a STO. Note if there is a safe stop availible on safety level this is to be used instead of the non safety signals. _
                   I_OFF1 := #Start,
                   I_OFF2 := "TRUE",
                   I_ResetFault := #I_AlarmResetPB,
                   I_BrakeRelease := #I_BrakeRelease,
                   I_ParameterSet := #I_ParameterSet,
                   I_SetpointSpeed := #SetpointSpeed,
                   I_Ramp := #RampToDrive,
                   C_HWSubInput := #C_HWSubInput,
                   C_HWSubInputStatus := #C_HWSubInputStatus,
                   C_HWSubOutput := #C_HWSubOutput,
                   C_DriveCurrent := #C_DriveCurrent,
                   C_MotorCurrent := #C_MotorCurrent,
                   O_DriveReady => #O_DriveReady,
                   O_OutputStageEnabled => #OutputStageEnabled,
                   O_MaintenanceSwitch => #MaintenanceSwitch,
                   O_ParameterSet => #O_ParameterSet,
                   O_PODataEnabled => #PODataEnabled,
                   O_Fault => #Fault,
                   O_Brake => #Brake,
                   O_ActorVoltageOverloadDO00 => #ActorVoltageOverloadDO00,
                   O_ActorVoltageOverloadDO01 => #ActorVoltageOverloadDO01,
                   O_ActorVoltageOverloadDO02 => #ActorVoltageOverloadDO02,
                   O_ActorVoltageOverloadDO03 => #ActorVoltageOverloadDO03,
                   O_SensorVoltageOverloadGroup1 => #SensorVoltageOverloadGroup1,
                   O_SensorVoltageOverloadGroup2 => #SensorVoltageOverloadGroup2,
                   O_SensorVoltageOverloadGroup3 => #SensorVoltageOverloadGroup3,
                   O_SensorVoltageOverloadGroup4 => #SensorVoltageOverloadGroup4,
                   "O_Undervoltage24V-S" => #"Undervoltage24V-S",
                   "O_InverterVoltageNotApplied24V-P" => #"InverterVoltageNotApplied24V-P",
                   O_MOVIFITSystemFault => #MOVIFITSystemFault,
                   H_StatusWord1 => #"H_GBMotor2W2S-MoviFitFCPN".H_StatusWord1[1].H_Word,
                   H_StatusWord2 => #"H_GBMotor2W2S-MoviFitFCPN".H_StatusWord2[1].H_Word,
                   H_StatusWord3 => #"H_GBMotor2W2S-MoviFitFCPN".H_StatusWord3[1].H_Word,
                   H_ControlWord => #"H_GBMotor2W2S-MoviFitFCPN".H_ControlWord[1].H_Word,
                   H_SetpointSpeed => #"H_GBMotor2W2S-MoviFitFCPN".H_SetpointSpeed[1].H_Word,
                   H_SetpointSpeedProCent => #"H_GBMotor2W2S-MoviFitFCPN".H_SetpointSpeedProCent[1].H_Real,
                   H_SetpointRamp => "NotUsedInt",
                   H_ActualCurrentA => #"H_GBMotor2W2S-MoviFitFCPN".H_ActualCurrentA[1].H_Real,
                   H_ActualCurrentProCent => #"H_GBMotor2W2S-MoviFitFCPN".H_ActualCurrentProCent[1].H_Real,
                   H_ActualWarning => #"H_GBMotor2W2S-MoviFitFCPN".H_ActualWarning[1].H_Int,
                   H_ActualFault => #"H_GBMotor2W2S-MoviFitFCPN".H_ActualFault[1].H_Int);
   END_IF;
END_REGION

REGION Network 20: **** 8 - Outputs **** Output stage enabled
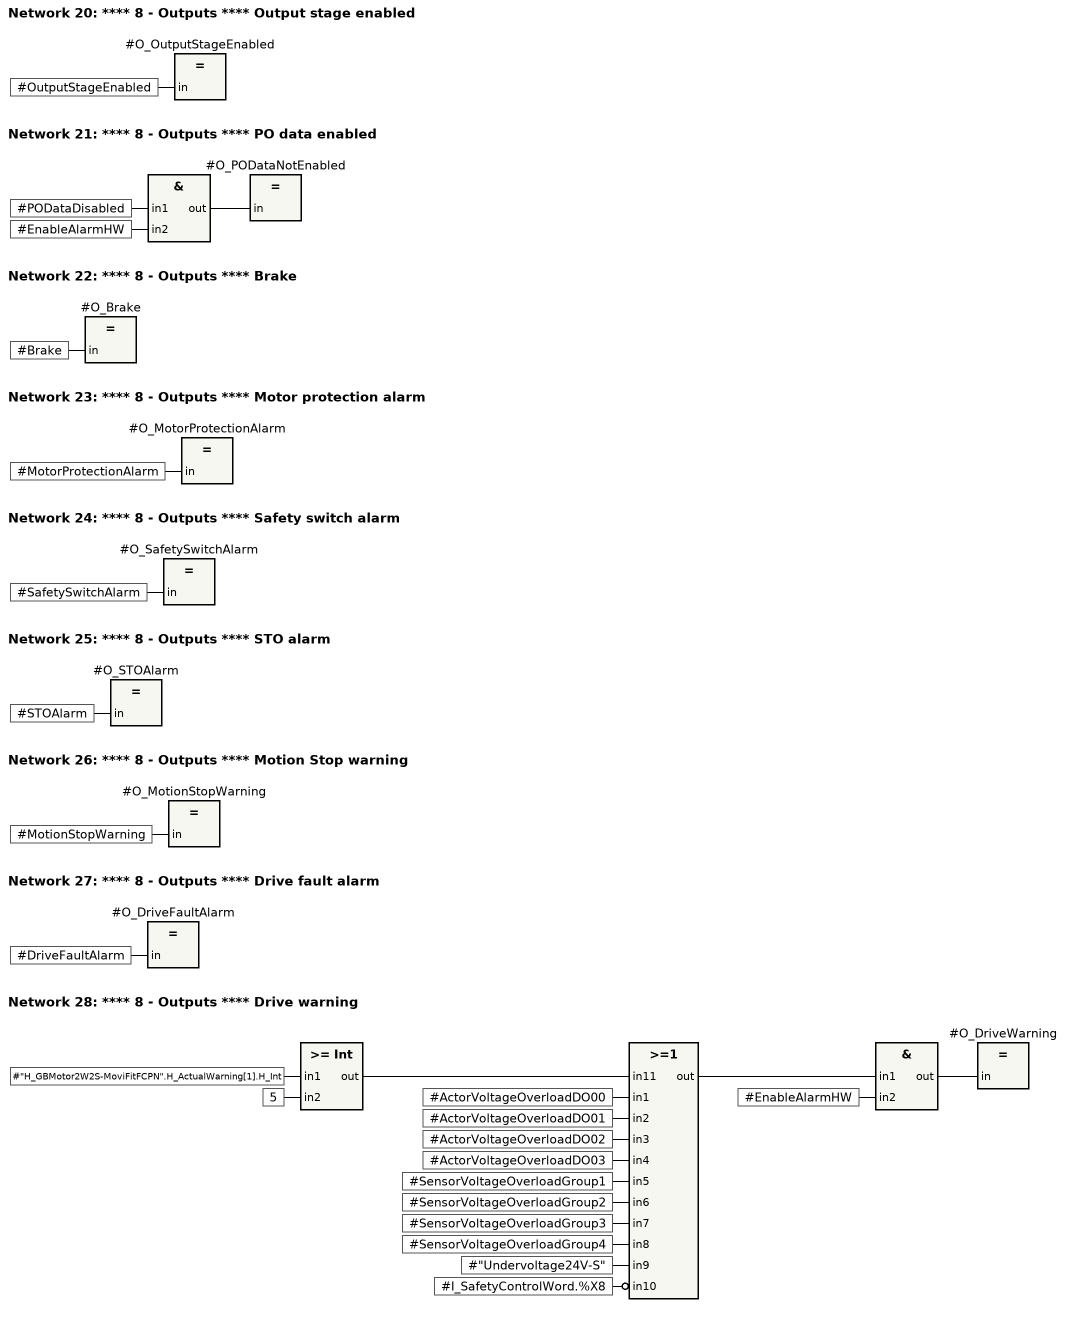
   #O_OutputStageEnabled := #OutputStageEnabled;
END_REGION

REGION Network 21: **** 8 - Outputs **** PO data enabled
   #O_PODataNotEnabled := #PODataDisabled AND #EnableAlarmHW;
END_REGION

REGION Network 22: **** 8 - Outputs **** Brake
   #O_Brake := #Brake;
END_REGION

REGION Network 23: **** 8 - Outputs **** Motor protection alarm
   // Motor protection alarm
   #O_MotorProtectionAlarm := #MotorProtectionAlarm;
END_REGION

REGION Network 24: **** 8 - Outputs **** Safety switch alarm
   // Safety switch alarm
   #O_SafetySwitchAlarm := #SafetySwitchAlarm;
END_REGION

REGION Network 25: **** 8 - Outputs **** STO alarm
   #O_STOAlarm := #STOAlarm;
END_REGION

REGION Network 26: **** 8 - Outputs **** Motion Stop warning
   #O_MotionStopWarning := #MotionStopWarning;
END_REGION

REGION Network 27: **** 8 - Outputs **** Drive fault alarm
   // Drive fault
   #O_DriveFaultAlarm := #DriveFaultAlarm;
END_REGION

REGION Network 28: **** 8 - Outputs **** Drive warning
   #O_DriveWarning := ((#"H_GBMotor2W2S-MoviFitFCPN".H_ActualWarning[1].H_Int >= 5) OR #ActorVoltageOverloadDO00 OR #ActorVoltageOverloadDO01 OR #ActorVoltageOverloadDO02 OR #ActorVoltageOverloadDO03 OR #SensorVoltageOverloadGroup1 OR #SensorVoltageOverloadGroup2 OR #SensorVoltageOverloadGroup3 OR #SensorVoltageOverloadGroup4 OR #"Undervoltage24V-S" OR NOT #I_SafetyControlWord.%X8) AND #EnableAlarmHW;
END_REGION

REGION Network 29: **** 8 - Outputs **** Config alarm
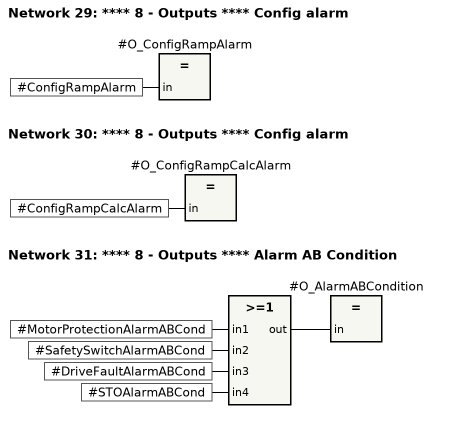
   #O_ConfigRampAlarm := #ConfigRampAlarm;
END_REGION

REGION Network 30: **** 8 - Outputs **** Config alarm
   #O_ConfigRampCalcAlarm := #ConfigRampCalcAlarm;
END_REGION

REGION Network 31: **** 8 - Outputs **** Alarm AB Condition
   // Alarm AB Condition
   #O_AlarmABCondition := #MotorProtectionAlarmABCond OR #SafetySwitchAlarmABCond OR #DriveFaultAlarmABCond OR #STOAlarmABCond;
END_REGION
END_FUNCTION_BLOCK
